TYPE T_RecipeStep : ST_RecipeStep; END_TYPE

(* stored: Version 1.1.0.1, ProductVersion 3.1.4024.15
   DUT T_RecipeStep: Id {14992e5c-b0af-4f2f-8472-d854a073721c} *)
